Fanuc KAREL source: KB00063.KL

PROGRAM KB00063
%NOLOCKGROUP
%ENVIRONMENT TPE
VAR
  P1: INTEGER
  P2: INTEGER
  P3: INTEGER
BEGIN
  P1 = 1
  P2 = 1
  P3 = 1
  DEL_INST_TPE(P1, P2, P3)
END KB00063
